// TIA Portal V18 export
// export: Created 2026-06-22T15:41:34.3740979Z, ExportSetting WithDefaults, DisplayName Totally Integrated Automation Portal, DisplayVersion V18, DisplayName TIA Portal Openness, DisplayVersion V18, DisplayName TIA Portal Version Control Interface, DisplayVersion V18, DisplayName STEP 7 Professional, DisplayVersion V18, DisplayName STEP 7 Safety, DisplayVersion V18, DisplayName WinCC Professional, DisplayVersion V18
DATA_BLOCK "DB1_NhanTuPLC1"   // DB1
{ S7_Optimized_Access := 'FALSE' }
VERSION : 0.1
// stored: AutoNumber true, IsOnlyStoredInLoadMemory false, IsWriteProtectedInAS false
   VAR
      Speed_SP_fromPLC1 : Real;
      Control_Byte : Bool;
      Reset_Cmd : Bool;
      DIR_Cmd : Bool;
   END_VAR
BEGIN
END_DATA_BLOCK
